INTERFACE IReadOnlyPointerUniqueSet EXTENDS ICollection

METHOD Contains : BOOL
VAR_INPUT
	element : PVOID;
END_VAR
END_METHOD

{attribute 'OPC.UA.DA.Property' := '1'}
{attribute 'monitoring' := 'call'}
PROPERTY ElementType : POINTER_TYPE
GET
END_GET
END_PROPERTY

METHOD GetByIndex : PVOID
VAR_INPUT
	index : DINT;
END_VAR
END_METHOD

END_INTERFACE

(* stored: Version 1.1.0.1
   Itf IReadOnlyPointerUniqueSet: Id {7a30d322-0ee6-0140-31b1-1a00871dabe8}
   Method Contains: Id {3ceaa5f6-d37f-0975-2a73-0d2f8d4dca87}
   Property ElementType: Id {ef8f627c-2345-037a-1cb1-698047520b24}
   Get Get: Id {a07d97cd-7500-07ce-321c-b914aa2a2786}
   Method GetByIndex: Id {9522a81b-725b-0af6-0700-b889e4d2baef} *)
